TYPE ST_Siemens_SendDp_Status :
STRUCT
	nSendBoolData			: WORD;
	nSendInt00				: INT;
	nSendInt01				: INT;
	nSendData				: WORD;
	nSendSequenceNumber		: WORD;
	nSendCrc				: WORD;
END_STRUCT
END_TYPE

(* stored: Version 1.1.0.1, ProductVersion 3.1.4024.12
   DUT ST_Siemens_SendDp_Status: Id {bb9bafd7-727e-0110-32b6-2d378cddfc74} *)
